{attribute 'global_init_slot' := '40001'}
PROGRAM LogList
VAR
	list: ARRAY[1..4000] OF T_MAXSTRING;
	lastlog: UINT := 1;
END_VAR

METHOD AddLog
VAR_INPUT
	text: T_MAXSTRING;
END_VAR
list[lastLog] := text;
lastLog := lastLog + 1;

IF lastLog = 4001 THEN
	lastLog := 1;
END_IF
END_METHOD

METHOD Print_To_ADS : DINT
VAR
	_counter : UINT := 1;
	_temp_string: T_MAXSTRING;
	_print_string: T_MAXSTRING;
	_error : DINT;
END_VAR
FOR _counter := 1 TO lastlog DO
	_temp_string := UINT_TO_ZEROSTRING(_counter);
	_temp_string := CONCAT(_temp_string, '  ');
	_temp_string := CONCAT(_temp_string, list[_counter]);
	_print_string := _temp_string;
	
	_error := ADSLOGSTR(ADSLOG_MSGTYPE_STRING, _print_string, '');
	
	IF _error <> 0 THEN
		Print_To_ADS := _error;
		RETURN;
	END_IF
END_FOR
END_METHOD

END_PROGRAM

(* stored: Version 1.1.0.1, ProductVersion 3.1.4024.12
   POU LogList: Id {c0015b5c-322e-41bb-a97b-a27bbf0ed492}, SpecialFunc None
   Method AddLog: Id {a2bba713-bb31-4ca0-92f4-c9d4114b1314}
   Method Print_To_ADS: Id {a8558cc6-5608-4256-b97b-96a99ae27a78} *)
